FUNCTION F_SyntaxError RETURNS BOOL
VAR_INPUT
END_VAR

END_FUNCTION

(* stored: Version 1.1.0.1, ProductVersion 3.1.4024.11
   POU F_SyntaxError: Id {245635d7-7d54-4aa8-92df-775383b63265}, SpecialFunc None *)
